// Mitsubishi GX Works2 project: combined data resister   PLC: FX1N/FX1NC

PROGRAM MAIN
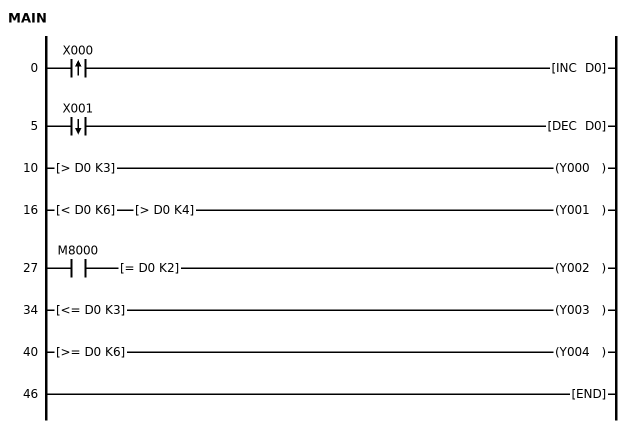
0     LDP     X000
      INC     D0
5     LDF     X001
      DEC     D0
10    LD>     D0 K3
      OUT     Y000
16    LD<     D0 K6
      AND>    D0 K4
      OUT     Y001
27    LD      M8000
      AND=    D0 K2
      OUT     Y002
34    LD<=    D0 K3
      OUT     Y003
40    LD>=    D0 K6
      OUT     Y004
46    END
END_PROGRAM
